// TIA Portal project "Project1" (V20)

(* hardware
DEVICE "S7-1200 station_1"  S7-1200 Station
   slot 0: "Rack_0"  S7-1200 Rack  Rack  V1.0
   slot 1: "PLC_1"  CPU 1215C DC/DC/Rly  6ES7 215-1HG40-0XB0  V4.6
DEVICE "HMI_1"  KTP700 Basic PN
   slot 0: "HMI_1"  KTP700 Basic PN  6AV2 123-2GB03-0AX0  17.0.0.0
   slot 1: "HMI_RT_1"  KTP700 Basic PN  6AV2 123-2GB03-0AX0  17.0.0.0
   slot 5: "HMI_1.IE_CP_1"  PROFINET Interface  17.0.0.0
      slot 1: "PROFINET Interface_1"  PROFINET Interface
         slot 1: "Port_1"  Port
*)

// ===== PLC "PLC_1"  CPU 1215C DC/DC/Rly =====

VAR_GLOBAL   // PLC tag table "Default tag table"
   "Auto" AT %I0.0 : Bool;
   "Manual" AT %I0.1 : Bool;
   "No Mode" AT %I0.2 : Bool;
   "Bottle Sensor" AT %I0.3 : Bool;
   "S1 PB" AT %I0.4 : Bool;
   "S2 PB" AT %I0.5 : Bool;
   "S3 PB" AT %I0.6 : Bool;
   "S4 PB" AT %I0.7 : Bool;
   "Mixer PB" AT %I1.0 : Bool;
   "Weight" AT %IW64 : Int;
   "S1" AT %Q0.0 : Bool;
   "S2" AT %Q0.1 : Bool;
   "S3" AT %Q0.2 : Bool;
   "S4" AT %Q0.3 : Bool;
   "Mixer" AT %Q0.4 : Bool;
   "close" AT %M0.0 : Bool;
END_VAR

DATA_BLOCK "bottle_main_1_DB"   // DB2
{ S7_Optimized_Access := 'TRUE' }
VERSION : 0.1
// stored: InstanceOfName bottle_main_1
"bottle_main_1"
BEGIN
END_DATA_BLOCK

DATA_BLOCK "tagsforproject_1"   // DB5
{ S7_Optimized_Access := 'TRUE' }
VERSION : 0.1
   VAR
      auto : Bool;
      manual : Bool;
      "no mode" : Bool;
      "bottle sensor" : Bool;
      "s1 pb" : Bool;
      "s2 pb" : Bool;
      "s3 pb" : Bool;
      "s4 pb" : Bool;
      "mixer pb" : Bool;
      "s1 out" : Bool;
      "s2 out" : Bool;
      "s3 out" : Bool;
      "s4 out" : Bool;
      "mixer out" : Bool;
      "weight indication" : Int;
      "S1 auto outpuut" : Bool;
      "S2 auto output" : Bool;
      "S3 auto output" : Bool;
      "S4 auto output" : Bool;
      "Mixer auto output" : Bool;
      autoruning : Bool;
      Ptrig1 : Bool;
      startrefill : Bool;
      Ptrig2 : Bool;
      Negative_edge_1 : Bool;
      Negative_edge_2 : Bool;
      Negative_edge_3 : Bool;
      Negative_edge_4 : Bool;
      Fill_is_ready : Bool;
      Stop_bottle_refill : Bool;
      Negative_edge_5 : Bool;
      start_refill_again : Bool;
      Ptrig : Bool;
      nomd : Bool;
      stop_refill : Bool;
   END_VAR
BEGIN
END_DATA_BLOCK

DATA_BLOCK "auto mode_DB"   // DB6
{ S7_Optimized_Access := 'TRUE' }
VERSION : 0.1
// stored: InstanceOfName auto mode
"auto mode"
BEGIN
END_DATA_BLOCK

DATA_BLOCK "Manual Mode_DB"   // DB7
{ S7_Optimized_Access := 'TRUE' }
VERSION : 0.1
// stored: InstanceOfName Manual Mode
"Manual Mode"
BEGIN
END_DATA_BLOCK

DATA_BLOCK "No mode process_DB"   // DB8
{ S7_Optimized_Access := 'TRUE' }
VERSION : 0.1
// stored: InstanceOfName No mode process
"No mode process"
BEGIN
END_DATA_BLOCK

DATA_BLOCK "IOs_Mapping_DB"   // DB9
{ S7_Optimized_Access := 'TRUE' }
VERSION : 0.1
// stored: InstanceOfName IOs_Mapping
"IOs_Mapping"
BEGIN
END_DATA_BLOCK

// folder: System blocks/Program resources

DATA_BLOCK "delay_auto"   // DB10
{ S7_Optimized_Access := 'TRUE' }
AUTHOR : Simatic
FAMILY : IEC
NAME : IEC_TMR
VERSION : 1.0
// stored: InstanceOfName IEC_TIMER
"IEC_TIMER"
BEGIN
END_DATA_BLOCK

DATA_BLOCK "apple_juice_pulse"   // DB11
{ S7_Optimized_Access := 'TRUE' }
AUTHOR : Simatic
FAMILY : IEC
NAME : IEC_TMR
VERSION : 1.0
// stored: InstanceOfName IEC_TIMER
"IEC_TIMER"
BEGIN
END_DATA_BLOCK

DATA_BLOCK "orange_juice_pulse"   // DB12
{ S7_Optimized_Access := 'TRUE' }
AUTHOR : Simatic
FAMILY : IEC
NAME : IEC_TMR
VERSION : 1.0
// stored: InstanceOfName IEC_TIMER
"IEC_TIMER"
BEGIN
END_DATA_BLOCK

DATA_BLOCK "lemon_juice_pulse"   // DB13
{ S7_Optimized_Access := 'TRUE' }
AUTHOR : Simatic
FAMILY : IEC
NAME : IEC_TMR
VERSION : 1.0
// stored: InstanceOfName IEC_TIMER
"IEC_TIMER"
BEGIN
END_DATA_BLOCK

DATA_BLOCK "Mixer_on"   // DB14
{ S7_Optimized_Access := 'TRUE' }
AUTHOR : Simatic
FAMILY : IEC
NAME : IEC_TMR
VERSION : 1.0
// stored: InstanceOfName IEC_TIMER
"IEC_TIMER"
BEGIN
END_DATA_BLOCK

// folder: (top level)

FUNCTION_BLOCK "bottle_main_1"   // FB1, LAD
{ S7_Optimized_Access := 'TRUE' }
VERSION : 0.1
BEGIN

REGION Network 1: auto
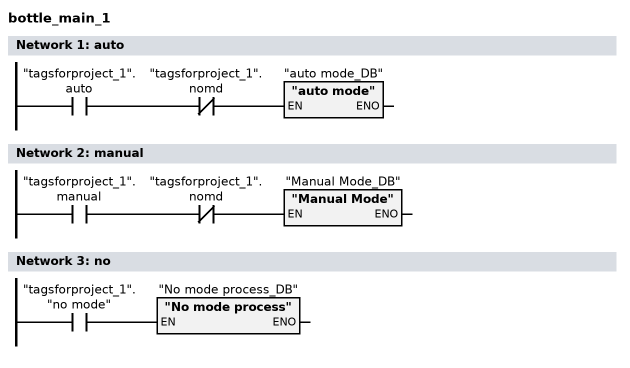
   RUNG wire#powerrail
      Contact( "tagsforproject_1".auto )
      I_Contact( "tagsforproject_1".nomd )
      "auto mode_DB"()
   END_RUNG
   // the same network as SCL:
   IF "tagsforproject_1".auto AND NOT "tagsforproject_1".nomd THEN
       "auto mode_DB"();   // "auto mode"
   END_IF;
END_REGION

REGION Network 2: manual
   RUNG wire#powerrail
      Contact( "tagsforproject_1".manual )
      I_Contact( "tagsforproject_1".nomd )
      "Manual Mode_DB"()
   END_RUNG
   // the same network as SCL:
   IF "tagsforproject_1".manual AND NOT "tagsforproject_1".nomd THEN
       "Manual Mode_DB"();   // "Manual Mode"
   END_IF;
END_REGION

REGION Network 3: no
   RUNG wire#powerrail
      Contact( "tagsforproject_1"."no mode" )
      "No mode process_DB"()
   END_RUNG
   // the same network as SCL:
   IF "tagsforproject_1"."no mode" THEN
       "No mode process_DB"();   // "No mode process"
   END_IF;
END_REGION
END_FUNCTION_BLOCK

FUNCTION_BLOCK "IOs_Mapping"   // FB2, LAD
{ S7_Optimized_Access := 'TRUE' }
VERSION : 0.1
BEGIN

REGION Network 1: inputs
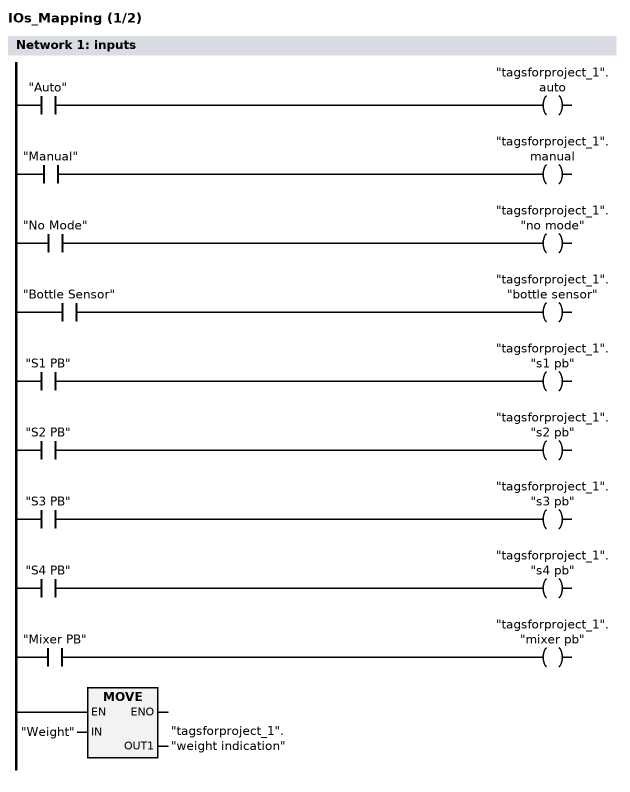
   RUNG wire#powerrail
      Contact( "Auto" )
      Coil( "tagsforproject_1".auto )
   END_RUNG
   RUNG wire#powerrail
      Contact( "Manual" )
      Coil( "tagsforproject_1".manual )
   END_RUNG
   RUNG wire#powerrail
      Contact( "No Mode" )
      Coil( "tagsforproject_1"."no mode" )
   END_RUNG
   RUNG wire#powerrail
      Contact( "Bottle Sensor" )
      Coil( "tagsforproject_1"."bottle sensor" )
   END_RUNG
   RUNG wire#powerrail
      Contact( "S1 PB" )
      Coil( "tagsforproject_1"."s1 pb" )
   END_RUNG
   RUNG wire#powerrail
      Contact( "S2 PB" )
      Coil( "tagsforproject_1"."s2 pb" )
   END_RUNG
   RUNG wire#powerrail
      Contact( "S3 PB" )
      Coil( "tagsforproject_1"."s3 pb" )
   END_RUNG
   RUNG wire#powerrail
      Contact( "S4 PB" )
      Coil( "tagsforproject_1"."s4 pb" )
   END_RUNG
   RUNG wire#powerrail
      Contact( "Mixer PB" )
      Coil( "tagsforproject_1"."mixer pb" )
   END_RUNG
   RUNG wire#powerrail
      Move(in := "Weight", out1 => "tagsforproject_1"."weight indication")
   END_RUNG
   // the same network as SCL:
   "tagsforproject_1".auto := "Auto";
   "tagsforproject_1".manual := "Manual";
   "tagsforproject_1"."no mode" := "No Mode";
   "tagsforproject_1"."bottle sensor" := "Bottle Sensor";
   "tagsforproject_1"."s1 pb" := "S1 PB";
   "tagsforproject_1"."s2 pb" := "S2 PB";
   "tagsforproject_1"."s3 pb" := "S3 PB";
   "tagsforproject_1"."s4 pb" := "S4 PB";
   "tagsforproject_1"."mixer pb" := "Mixer PB";
   "tagsforproject_1"."weight indication" := "Weight";
END_REGION

REGION Network 2: outputs
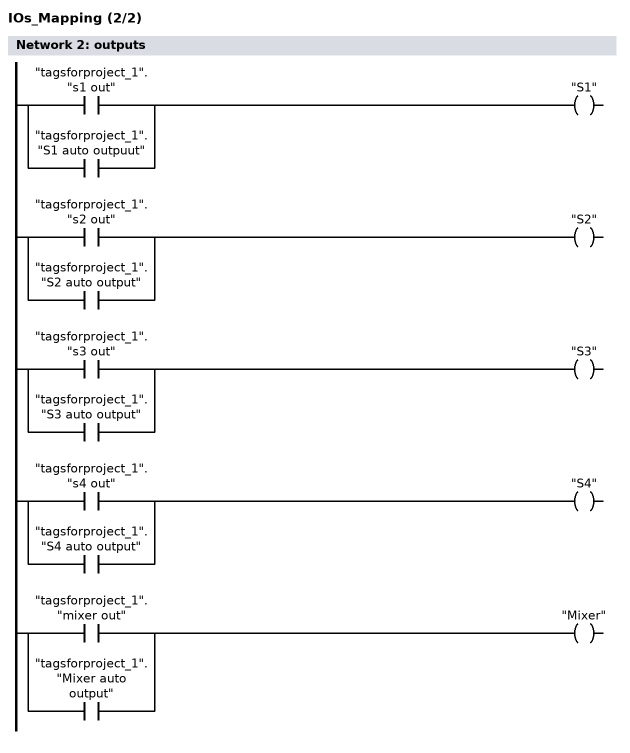
   RUNG wire#powerrail
      Contact( "tagsforproject_1"."s1 out" )
      wire#w1
      Coil( "S1" )
   END_RUNG
   RUNG wire#powerrail
      Contact( "tagsforproject_1"."S1 auto outpuut" )
   END_RUNG wire#w1
   RUNG wire#powerrail
      Contact( "tagsforproject_1"."s2 out" )
      wire#w2
      Coil( "S2" )
   END_RUNG
   RUNG wire#powerrail
      Contact( "tagsforproject_1"."S2 auto output" )
   END_RUNG wire#w2
   RUNG wire#powerrail
      Contact( "tagsforproject_1"."s3 out" )
      wire#w3
      Coil( "S3" )
   END_RUNG
   RUNG wire#powerrail
      Contact( "tagsforproject_1"."S3 auto output" )
   END_RUNG wire#w3
   RUNG wire#powerrail
      Contact( "tagsforproject_1"."s4 out" )
      wire#w4
      Coil( "S4" )
   END_RUNG
   RUNG wire#powerrail
      Contact( "tagsforproject_1"."S4 auto output" )
   END_RUNG wire#w4
   RUNG wire#powerrail
      Contact( "tagsforproject_1"."mixer out" )
      wire#w5
      Coil( "Mixer" )
   END_RUNG
   RUNG wire#powerrail
      Contact( "tagsforproject_1"."Mixer auto output" )
   END_RUNG wire#w5
   // the same network as SCL:
   "S1" := "tagsforproject_1"."s1 out" OR "tagsforproject_1"."S1 auto outpuut";
   "S2" := "tagsforproject_1"."s2 out" OR "tagsforproject_1"."S2 auto output";
   "S3" := "tagsforproject_1"."s3 out" OR "tagsforproject_1"."S3 auto output";
   "S4" := "tagsforproject_1"."s4 out" OR "tagsforproject_1"."S4 auto output";
   "Mixer" := "tagsforproject_1"."mixer out" OR "tagsforproject_1"."Mixer auto output";
END_REGION
END_FUNCTION_BLOCK

FUNCTION_BLOCK "Manual Mode"   // FB3, LAD
{ S7_Optimized_Access := 'TRUE' }
VERSION : 0.1
BEGIN

REGION Network 1
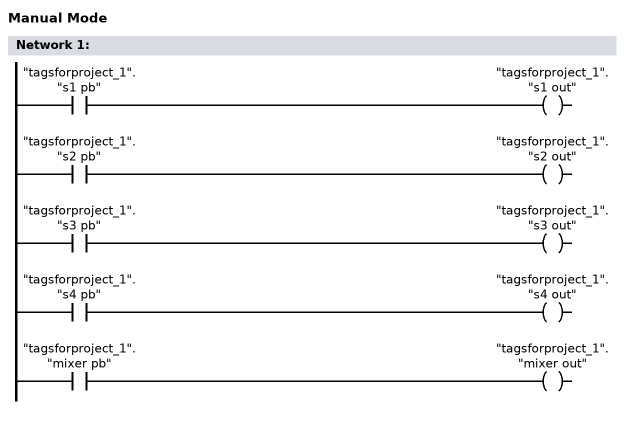
   RUNG wire#powerrail
      Contact( "tagsforproject_1"."s1 pb" )
      Coil( "tagsforproject_1"."s1 out" )
   END_RUNG
   RUNG wire#powerrail
      Contact( "tagsforproject_1"."s2 pb" )
      Coil( "tagsforproject_1"."s2 out" )
   END_RUNG
   RUNG wire#powerrail
      Contact( "tagsforproject_1"."s3 pb" )
      Coil( "tagsforproject_1"."s3 out" )
   END_RUNG
   RUNG wire#powerrail
      Contact( "tagsforproject_1"."s4 pb" )
      Coil( "tagsforproject_1"."s4 out" )
   END_RUNG
   RUNG wire#powerrail
      Contact( "tagsforproject_1"."mixer pb" )
      Coil( "tagsforproject_1"."mixer out" )
   END_RUNG
   // the same network as SCL:
   "tagsforproject_1"."s1 out" := "tagsforproject_1"."s1 pb";
   "tagsforproject_1"."s2 out" := "tagsforproject_1"."s2 pb";
   "tagsforproject_1"."s3 out" := "tagsforproject_1"."s3 pb";
   "tagsforproject_1"."s4 out" := "tagsforproject_1"."s4 pb";
   "tagsforproject_1"."mixer out" := "tagsforproject_1"."mixer pb";
END_REGION
END_FUNCTION_BLOCK

FUNCTION_BLOCK "auto mode"   // FB4, LAD
{ S7_Optimized_Access := 'TRUE' }
VERSION : 0.1
   VAR_TEMP   // added for the SCL form of the ladder/FBD networks
      _w1 : Bool;
      _w2 : Bool;
      _w3 : Bool;
      _w4 : Bool;
      _w5 : Bool;
      _w6 : Bool;
      _w7 : Bool;
   END_VAR
BEGIN

REGION Network 1
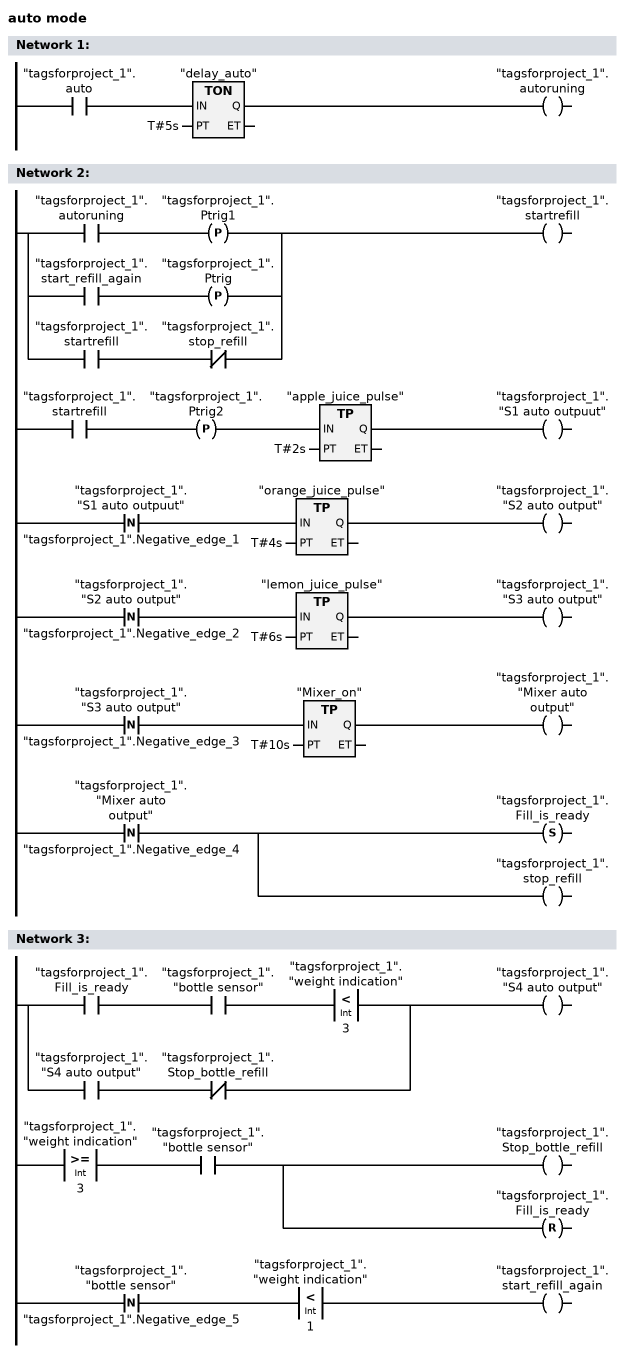
   "delay_auto".TON(IN := "tagsforproject_1".auto, PT := T#5s);
   "tagsforproject_1".autoruning := "delay_auto".Q;
END_REGION

REGION Network 2
   #_w1 := "tagsforproject_1".autoruning AND NOT "tagsforproject_1".Ptrig1;   // rising edge
   "tagsforproject_1".Ptrig1 := "tagsforproject_1".autoruning;
   #_w2 := "tagsforproject_1".start_refill_again AND NOT "tagsforproject_1".Ptrig;   // rising edge
   "tagsforproject_1".Ptrig := "tagsforproject_1".start_refill_again;
   "tagsforproject_1".startrefill := #_w1 OR #_w2 OR ("tagsforproject_1".startrefill AND NOT "tagsforproject_1".stop_refill);
   #_w3 := "tagsforproject_1".startrefill AND NOT "tagsforproject_1".Ptrig2;   // rising edge
   "tagsforproject_1".Ptrig2 := "tagsforproject_1".startrefill;
   "apple_juice_pulse".TP(IN := #_w3, PT := T#2s);
   "tagsforproject_1"."S1 auto outpuut" := "apple_juice_pulse".Q;
   #_w4 := NOT "tagsforproject_1"."S1 auto outpuut" AND "tagsforproject_1".Negative_edge_1;   // falling edge of "tagsforproject_1"."S1 auto outpuut"
   "tagsforproject_1".Negative_edge_1 := "tagsforproject_1"."S1 auto outpuut";
   "orange_juice_pulse".TP(IN := #_w4, PT := T#4s);
   "tagsforproject_1"."S2 auto output" := "orange_juice_pulse".Q;
   #_w5 := NOT "tagsforproject_1"."S2 auto output" AND "tagsforproject_1".Negative_edge_2;   // falling edge of "tagsforproject_1"."S2 auto output"
   "tagsforproject_1".Negative_edge_2 := "tagsforproject_1"."S2 auto output";
   "lemon_juice_pulse".TP(IN := #_w5, PT := T#6s);
   "tagsforproject_1"."S3 auto output" := "lemon_juice_pulse".Q;
   #_w6 := NOT "tagsforproject_1"."S3 auto output" AND "tagsforproject_1".Negative_edge_3;   // falling edge of "tagsforproject_1"."S3 auto output"
   "tagsforproject_1".Negative_edge_3 := "tagsforproject_1"."S3 auto output";
   "Mixer_on".TP(IN := #_w6, PT := T#10s);
   "tagsforproject_1"."Mixer auto output" := "Mixer_on".Q;
   #_w7 := NOT "tagsforproject_1"."Mixer auto output" AND "tagsforproject_1".Negative_edge_4;   // falling edge of "tagsforproject_1"."Mixer auto output"
   "tagsforproject_1".Negative_edge_4 := "tagsforproject_1"."Mixer auto output";
   IF #_w7 THEN "tagsforproject_1".Fill_is_ready := TRUE; END_IF;
   "tagsforproject_1".stop_refill := #_w7;
END_REGION

REGION Network 3
   RUNG wire#powerrail
      Contact( "tagsforproject_1".Fill_is_ready )
      Contact( "tagsforproject_1"."bottle sensor" )
      { S7_Templates := "SrcType := Int" } LT_Contact(in1 := "tagsforproject_1"."weight indication", in2 := 3)
      wire#w1
      Coil( "tagsforproject_1"."S4 auto output" )
   END_RUNG
   RUNG wire#powerrail
      Contact( "tagsforproject_1"."S4 auto output" )
      I_Contact( "tagsforproject_1".Stop_bottle_refill )
   END_RUNG wire#w1
   RUNG wire#powerrail
      { S7_Templates := "SrcType := Int" } GE_Contact(in1 := "tagsforproject_1"."weight indication", in2 := 3)
      Contact( "tagsforproject_1"."bottle sensor" )
      wire#w2
      Coil( "tagsforproject_1".Stop_bottle_refill )
   END_RUNG
   RUNG wire#w2
      R_Coil( "tagsforproject_1".Fill_is_ready )
   END_RUNG
   RUNG wire#powerrail
      N_Contact(operand := "tagsforproject_1"."bottle sensor", bit := "tagsforproject_1".Negative_edge_5)
      { S7_Templates := "SrcType := Int" } LT_Contact(in1 := "tagsforproject_1"."weight indication", in2 := 1)
      Coil( "tagsforproject_1".start_refill_again )
   END_RUNG
   // the same network as SCL:
   "tagsforproject_1"."S4 auto output" := ("tagsforproject_1".Fill_is_ready AND "tagsforproject_1"."bottle sensor" AND ("tagsforproject_1"."weight indication" < 3)) OR ("tagsforproject_1"."S4 auto output" AND NOT "tagsforproject_1".Stop_bottle_refill);
   "tagsforproject_1".Stop_bottle_refill := ("tagsforproject_1"."weight indication" >= 3) AND "tagsforproject_1"."bottle sensor";
   IF "tagsforproject_1".Stop_bottle_refill THEN "tagsforproject_1".Fill_is_ready := FALSE; END_IF;
   #_w1 := NOT "tagsforproject_1"."bottle sensor" AND "tagsforproject_1".Negative_edge_5;   // falling edge of "tagsforproject_1"."bottle sensor"
   "tagsforproject_1".Negative_edge_5 := "tagsforproject_1"."bottle sensor";
   "tagsforproject_1".start_refill_again := #_w1 AND ("tagsforproject_1"."weight indication" < 1);
END_REGION
END_FUNCTION_BLOCK

FUNCTION_BLOCK "No mode process"   // FB5, LAD
{ S7_Optimized_Access := 'TRUE' }
VERSION : 0.1
BEGIN

REGION Network 1
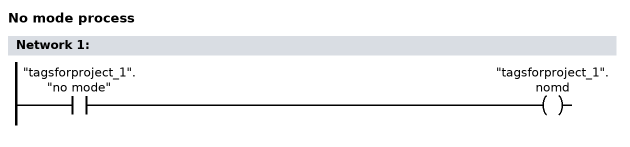
   RUNG wire#powerrail
      Contact( "tagsforproject_1"."no mode" )
      Coil( "tagsforproject_1".nomd )
   END_RUNG
   // the same network as SCL:
   "tagsforproject_1".nomd := "tagsforproject_1"."no mode";
END_REGION
END_FUNCTION_BLOCK

ORGANIZATION_BLOCK "Main"   // OB1, LAD, ProgramCycle
TITLE = "Main Program Sweep (Cycle)"
{ S7_Optimized_Access := 'TRUE' }
VERSION : 0.1
   VAR_INPUT
      Initial_Call : Bool;   // Initial call of this OB
      Remanence : Bool;   // =True, if remanent data are available
   END_VAR
   VAR_TEMP
      e_time_2 : Time;
      count : Int;
   END_VAR
BEGIN

REGION Network 1
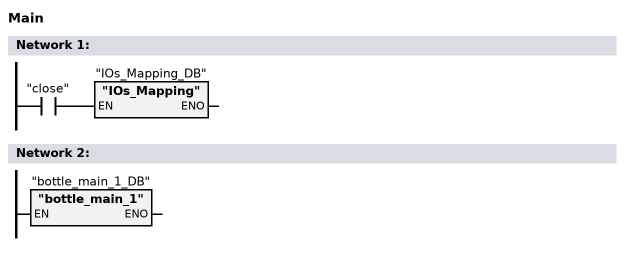
   RUNG wire#powerrail
      Contact( "close" )
      "IOs_Mapping_DB"()
   END_RUNG
   // the same network as SCL:
   IF "close" THEN
       "IOs_Mapping_DB"();   // "IOs_Mapping"
   END_IF;
END_REGION

REGION Network 2
   RUNG wire#powerrail
      "bottle_main_1_DB"()
   END_RUNG
   // the same network as SCL:
   "bottle_main_1_DB"();   // "bottle_main_1"
END_REGION
END_ORGANIZATION_BLOCK

(* ===== HMI "HMI_RT_1" =====
connection "HMI_Connection_1": ETHERNET, SMART_S7_1200_OMS

screen "Screen_2" 800x480
   Button "Button_1" at 131,67 size 96x32; TextOff 'Text'
   Button "Button_2" at 262,78 size 96x32; TextOff 'Text'
   Button "Button_3" at 431,91 size 96x32; TextOff 'Text'
   Button "Button_4" at 537,88 size 96x32; TextOff 'Text'
*)